// TwinCAT 3 PLC project Plc
// ProgramVersion: 3.1.4024.0
// libraries:
//   Tc2_Standard, * (Beckhoff Automation GmbH)
//   Tc2_System, * (Beckhoff Automation GmbH)
//   Tc3_Module, * (Beckhoff Automation GmbH)
//   VisuSymbols,3.5.10.0,System
// project tree:
//   DUTs/ E_States.TcDUT
//   / Gestore di visualizzazione.TcVMO (not stored), GlobalTextList.TcGTLO, PlcTask.TcTTO
//   GVLs/ GVL.TcGVL
//   POUs/ FB_StateMachine.TcPOU, FB_Visualization.TcPOU, MAIN.TcPOU
//   VISUs/ Visualization.TcVIS
// real-time tasks:
//   TASK PlcTask: cycle T#10ms, priority 20, ADS port 350

CONFIGURATION Plc
    RESOURCE PLC ON TwinCAT3
        TASK PlcTask(INTERVAL := T#10ms, PRIORITY := 20);
        PROGRAM MAIN WITH PlcTask : MAIN;
    END_RESOURCE
END_CONFIGURATION

// ---- DUTs/E_States.TcDUT
{attribute 'qualified_only'}
{attribute 'strict'}
TYPE E_States :
(
	eStop := 0,
	eMovingLeft,
	eMovingRight,
	eLoad,
	eUnload
);
END_TYPE

// ---- GVLs/GVL.TcGVL
{attribute 'qualified_only'}
VAR_GLOBAL
	//Input
	bStart : BOOL;
	bStop : BOOL;
	bSensorLeft : BOOL;
	bLimitLeft : BOOL;
	bLimitRight : BOOL;
	
	//Output
	bMotorLeft : BOOL;
	bMotorRight : BOOL;
END_VAR

// ---- POUs/MAIN.TcPOU
PROGRAM MAIN
VAR
	StateMachine: FB_StateMachine;
	Visualization: FB_Visualization;
END_VAR

StateMachine(bStart:= GVL.bStart, bStop:= GVL.bStop, bLimitLeft:= GVL.bLimitLeft, bLimitRight:= GVL.bLimitRight );
Visualization(bMovingRight:= StateMachine.bMovingRight, bMovingLeft:=StateMachine.bMovingLeft);
GVL.bLimitLeft := Visualization.bLimitLeft;
GVL.bLimitRight := Visualization.bLimitRight;

END_PROGRAM

// ---- POUs/FB_StateMachine.TcPOU
FUNCTION_BLOCK FB_StateMachine
VAR_INPUT
	bStart : BOOL;
	bStop : BOOL;
	bLimitLeft : BOOL;
	bLimitRight: BOOL;
END_VAR
VAR_OUTPUT
	bMovingRight : BOOL;
	bMovingLeft: BOOL;
END_VAR
VAR
	TrigStop: R_TRIG;
	state : E_States;
	prevState : E_States;
	sState: STRING;
END_VAR

TrigStop(CLK:=bStop);

IF TrigStop.Q THEN
	prevState := state;
	state:= E_States.eStop;
END_IF	


CASE state OF
	E_States.eStop:
		sState := 'Stop';
		bMovingRight := FALSE;
		bMovingLeft := FALSE;
		IF bStart THEN
			IF prevState = E_States.eMovingLeft THEN
				state:= E_States.eMovingLeft;
			ELSE
				state:= E_States.eMovingRight;
			END_IF
		END_IF
	
	E_States.eMovingRight:
		sState := 'Moving Right';
		bMovingRight := TRUE;
		bMovingLeft := FALSE;
		IF bLimitRight THEN
			state:= E_States.eMovingLeft;
		END_IF
	
	E_States.eMovingLeft:
		sState := 'Moving Left';
		bMovingRight := FALSE;
		bMovingLeft := TRUE;
		IF bLimitLeft THEN
			state:= E_States.eMovingRight;
		END_IF
	
	
END_CASE

END_FUNCTION_BLOCK

// ---- POUs/FB_Visualization.TcPOU
FUNCTION_BLOCK FB_Visualization
VAR_INPUT
	bMovingRight : BOOL;
	bMovingLeft : BOOL;
END_VAR
VAR_OUTPUT
	bLimitLeft : BOOL;
	bLimitRight: BOOL;
END_VAR
VAR
	Position: REAL;
END_VAR

IF bMovingRight THEN
	bLimitLeft := FALSE;
	bLimitRight := FALSE;
	Position := Position + 0.5;
	IF (Position >= 310) THEN
		bLimitRight := TRUE;
	END_IF
ELSIF bMovingLeft THEN
	bLimitLeft := FALSE;
	bLimitRight := FALSE;
	Position := Position - 0.5;
	IF (Position <=  0) THEN
		bLimitLeft := TRUE;
	END_IF
END_IF

END_FUNCTION_BLOCK

// ---- GlobalTextList.TcGTLO
TEXTLIST GlobalTextList
  563 = '%s'
  498 = 'START'
  690 = 'STOP'
END_TEXTLIST

// ---- VISUs/Visualization.TcVIS
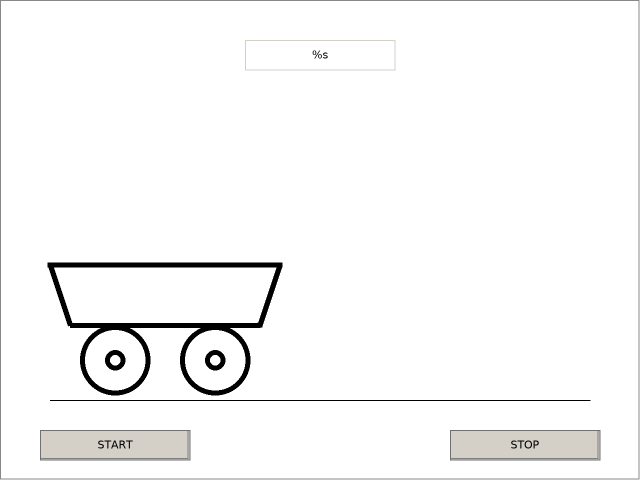
VISUALIZATION Visualization  // 640x480
    Line (50,400) (590,400)
    Group (50,265 230x130)
        p3560616238: MAIN.Visualization.Position
        Ellipse (30,60 70x70)
        Ellipse (55,85 20x20)
        Ellipse (130,60 70x70)
        Ellipse (155,85 20x20)
        Polyline (20,60) (210,60) (230,0) (0,0) (20,60)
    Button (40,430 150x30), "START"
        tap GVL.bStart
    Button (450,430 150x30), "STOP"
        tap GVL.bStop
    Textfield (245,40 150x30), "%s", text variable: MAIN.StateMachine.sState
END_VISUALIZATION
